{attribute 'qualified_only'}
{attribute 'strict'}
{attribute 'to_string'}

TYPE eBreakerOperationMode :
(
	none 				:= 0,
	GridFeedthrough		:= 1,
	ExtGrid				:= 2,
	GenDroop			:= 3,
	GenIso				:= 4,
	GenFix				:= 5
);
END_TYPE

(* stored: Version 1.1.0.1, ProductVersion 3.1.4026.18
   DUT eBreakerOperationMode: Id {529cc822-dd52-46d6-925c-3cc544641e20} *)
